// SIMATIC S7-200 SMART project (STEP 7-Micro/WIN SMART), CPU SR30

SYMBOL_TABLE 风机和阀
温度量程下限           VD232
温度量程上限           VD228
压力量程下限           VD324
压力量程上限           VD328
风机停止             V2.0
风机启动             V2.1
风机远程             V2.2
风机故障             V2.3
风机输出             V2.4
风机               V2.5
风机运行反馈           V2.6
风机超时             V2.7
阀1停止             V3.0
阀1启动             V3.1
阀1远程             V3.2
阀1故障             V3.3
阀1输出             V3.4
阀1               V3.5
阀1运行反馈           V3.6
阀1超时             V3.7
阀2停止             V4.0
阀2启动             V4.1
阀2远程             V4.2
阀2故障             V4.3
阀2输出             V4.4
阀2               V4.5
阀2运行反馈           V4.6
阀2超时             V4.7
阀3停止             V5.0
阀3启动             V5.1
阀3远程             V5.2
阀3故障             V5.3
阀3输出             V5.4
阀3               V5.5
阀3运行反馈           V5.6
阀3超时             V5.7
阀4停止             V6.0
阀4启动             V6.1
阀4远程             V6.2
阀4故障             V6.3
阀4输出             V6.4
阀4               V6.5
阀4运行反馈           V6.6
阀4超时             V6.7
END_SYMBOL_TABLE

SYMBOL_TABLE 系统符号
Always_On        SM0.0    // 始终接通
END_SYMBOL_TABLE

SYMBOL_TABLE 点火烧嘴
急停               V10.7
点亮屏幕             V11.1
故障码              VW200
高温报警             V11.2
低温报警             V11.3
流量高报警            V11.4
流量低报警            V11.5
点火命令1            V7.0
点火成功信号1          V7.1
故障复位             V7.2
点火变压器1           V7.3
点火电磁阀1           V7.4
报警1              V7.5
空气压力1            V9.0
燃气压力1            V9.1
燃气泄漏             V9.2
允许点火1            V9.3
本地               V9.4
远程               V9.5
灯光报警1            V10.1
消音自锁             V10.2
声响报警1            V10.3
消音命令             V10.4
点火命令2            V7.6
点火成功信号2          V7.7
点火变压器2           V8.1
点火电磁阀2           V8.2
报警2              V8.3
空气压力2            V9.6
燃气压力2            V9.7
允许点火2            V10.0
灯光报警2            V10.5
声响报警2            V10.6
END_SYMBOL_TABLE

ORGANIZATION_BLOCK MAIN:OB1
TITLE=程序注释
BEGIN
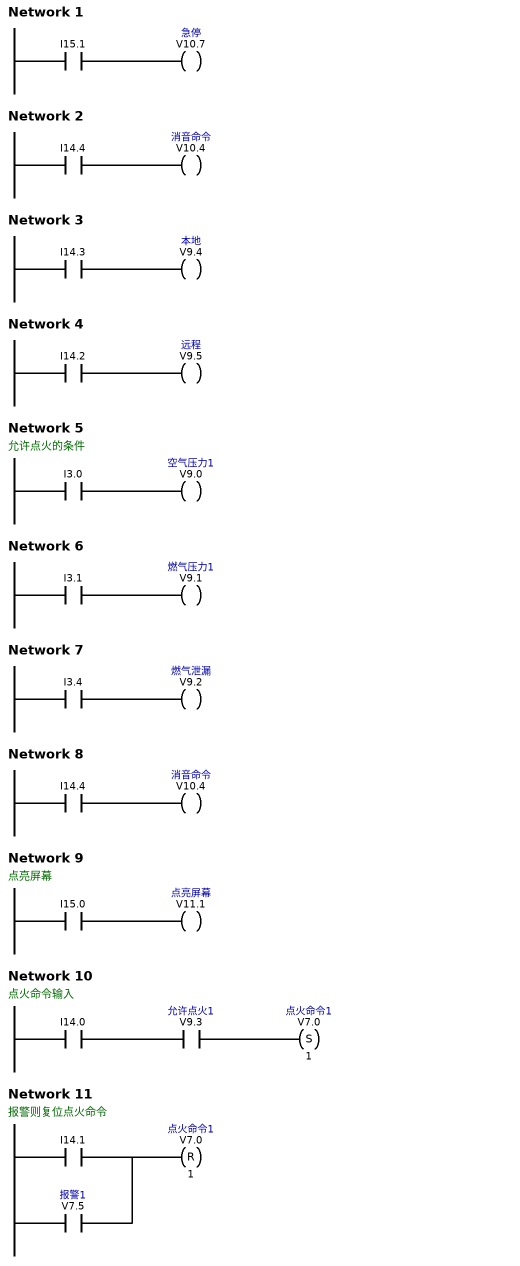
Network 1
LD     I15.1
=      急停:V10.7
Network 2
LD     I14.4
=      消音命令:V10.4
Network 3
LD     I14.3
=      本地:V9.4
Network 4
LD     I14.2
=      远程:V9.5
Network 5
// 允许点火的条件
LD     I3.0
=      空气压力1:V9.0
Network 6
LD     I3.1
=      燃气压力1:V9.1
Network 7
LD     I3.4
=      燃气泄漏:V9.2
Network 8
LD     I14.4
=      消音命令:V10.4
Network 9
// 点亮屏幕
LD     I15.0
=      点亮屏幕:V11.1
Network 10
// 点火命令输入
LD     I14.0
A      允许点火1:V9.3
S      点火命令1:V7.0, 1
Network 11
// 报警则复位点火命令
LD     I14.1
O      报警1:V7.5
R      点火命令1:V7.0, 1
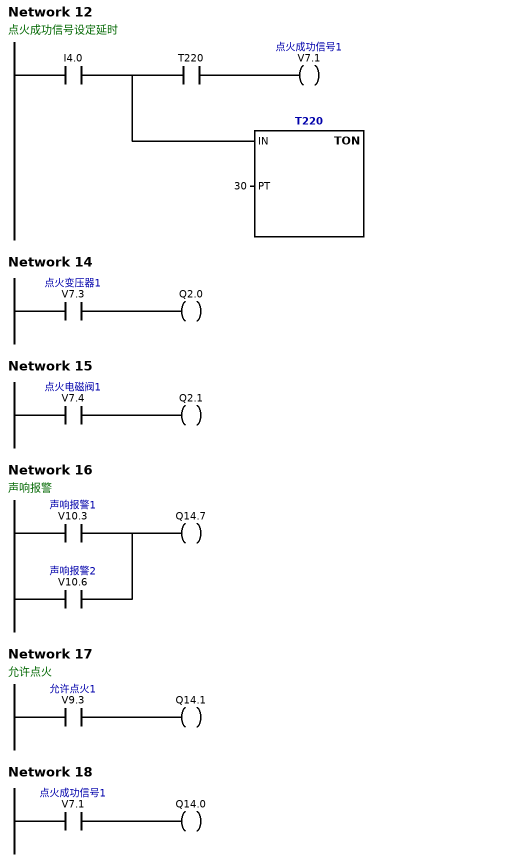
Network 12
// 点火成功信号设定延时
LD     I4.0
LPS
A      T220
=      点火成功信号1:V7.1
LPP
TON    T220, 30
Network 14
LD     点火变压器1:V7.3
=      Q2.0
Network 15
LD     点火电磁阀1:V7.4
=      Q2.1
Network 16
// 声响报警
LD     声响报警1:V10.3
O      声响报警2:V10.6
=      Q14.7
Network 17
// 允许点火
LD     允许点火1:V9.3
=      Q14.1
Network 18
LD     点火成功信号1:V7.1
=      Q14.0
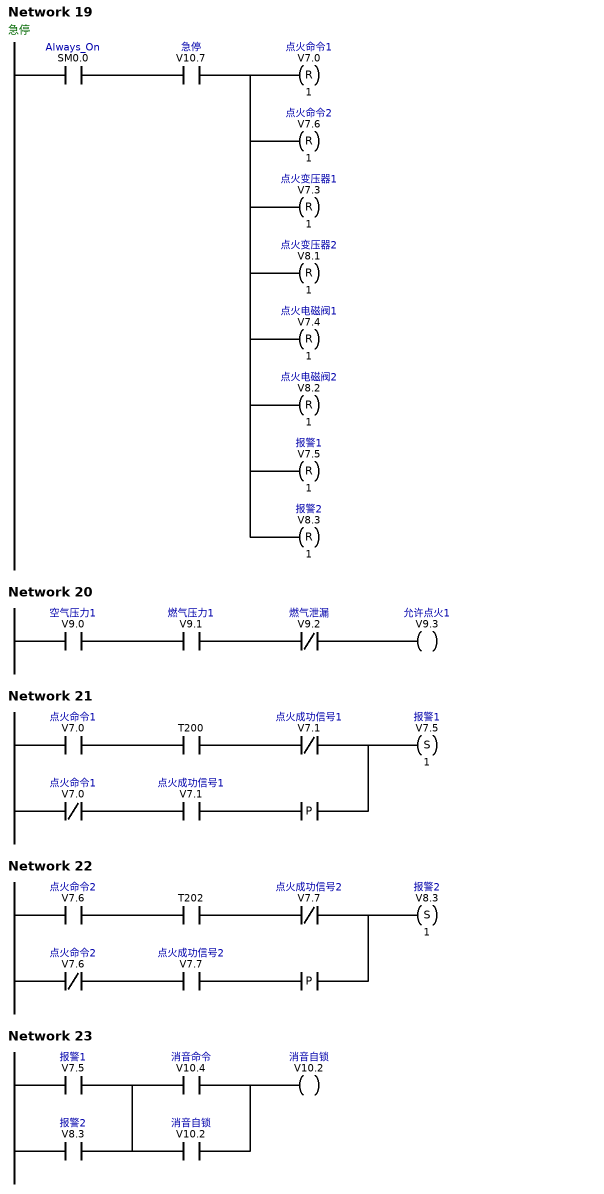
Network 19
// 急停
LD     Always_On:SM0.0
A      急停:V10.7
R      点火命令1:V7.0, 1
R      点火命令2:V7.6, 1
R      点火变压器1:V7.3, 1
R      点火变压器2:V8.1, 1
R      点火电磁阀1:V7.4, 1
R      点火电磁阀2:V8.2, 1
R      报警1:V7.5, 1
R      报警2:V8.3, 1
Network 20
LD     空气压力1:V9.0
A      燃气压力1:V9.1
AN     燃气泄漏:V9.2
=      允许点火1:V9.3
Network 21
LD     点火命令1:V7.0
A      T200
AN     点火成功信号1:V7.1
LDN    点火命令1:V7.0
A      点火成功信号1:V7.1
EU
OLD
S      报警1:V7.5, 1
Network 22
LD     点火命令2:V7.6
A      T202
AN     点火成功信号2:V7.7
LDN    点火命令2:V7.6
A      点火成功信号2:V7.7
EU
OLD
S      报警2:V8.3, 1
Network 23
LD     报警1:V7.5
O      报警2:V8.3
LD     消音命令:V10.4
O      消音自锁:V10.2
ALD
=      消音自锁:V10.2
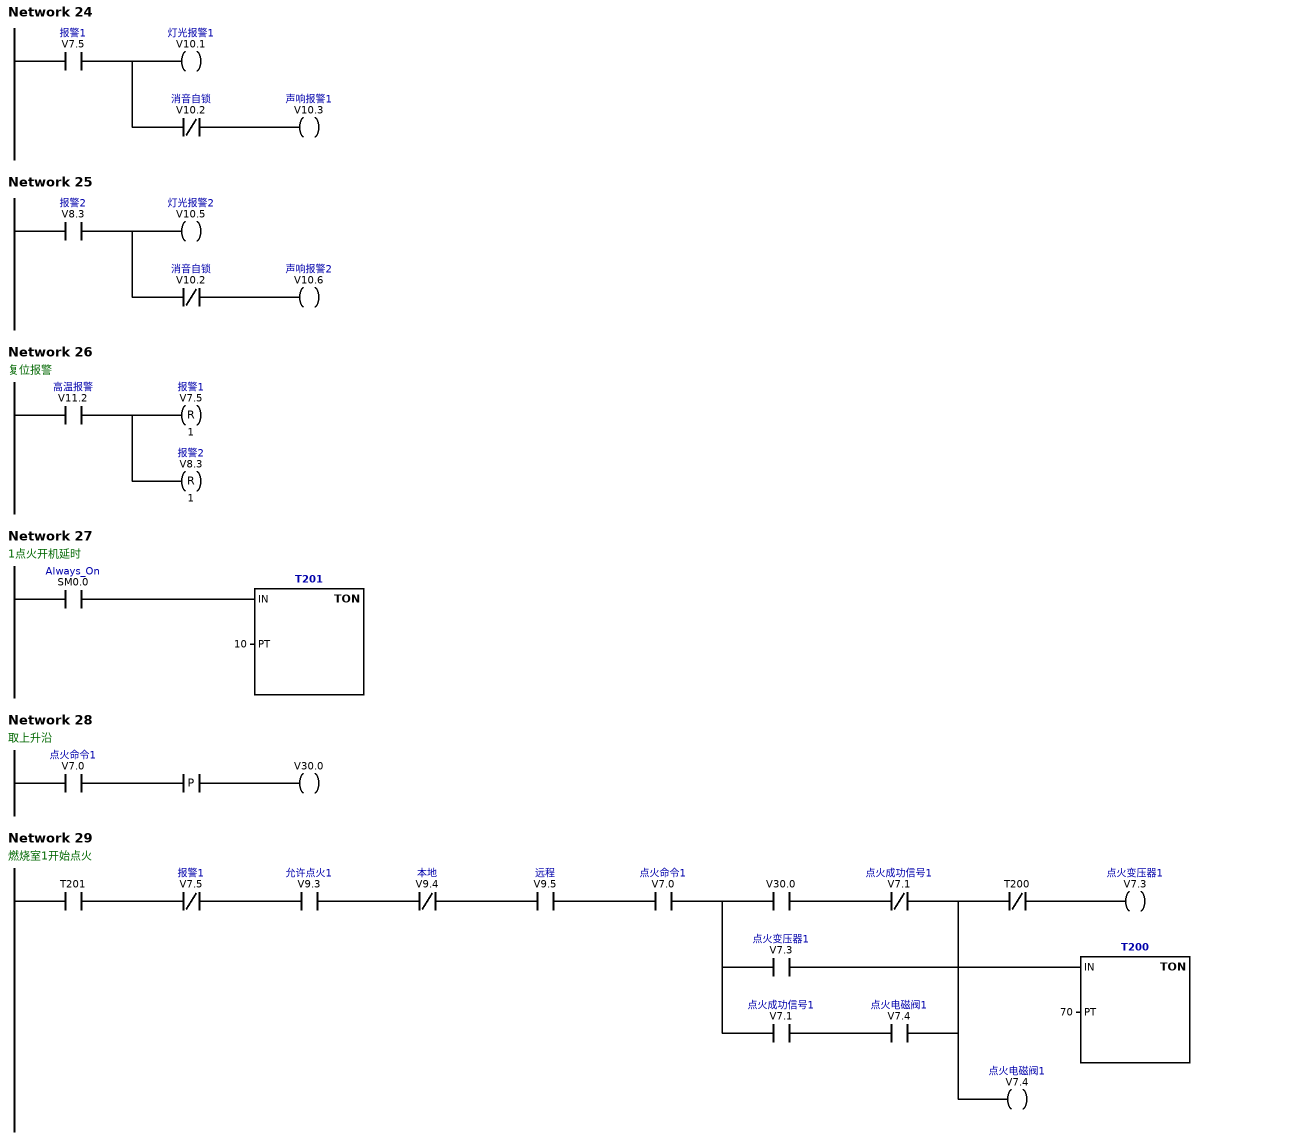
Network 24
LD     报警1:V7.5
=      灯光报警1:V10.1
AN     消音自锁:V10.2
=      声响报警1:V10.3
Network 25
LD     报警2:V8.3
=      灯光报警2:V10.5
AN     消音自锁:V10.2
=      声响报警2:V10.6
Network 26
// 复位报警
LD     高温报警:V11.2
R      报警1:V7.5, 1
R      报警2:V8.3, 1
Network 27
// 1点火开机延时
LD     Always_On:SM0.0
TON    T201, 10
Network 28
// 取上升沿
LD     点火命令1:V7.0
EU
=      V30.0
Network 29
// 燃烧室1开始点火
LD     T201
AN     报警1:V7.5
A      允许点火1:V9.3
AN     本地:V9.4
A      远程:V9.5
A      点火命令1:V7.0
LD     V30.0
AN     点火成功信号1:V7.1
O      点火变压器1:V7.3
LD     点火成功信号1:V7.1
A      点火电磁阀1:V7.4
OLD
ALD
LPS
AN     T200
=      点火变压器1:V7.3
LRD
TON    T200, 70
LPP
=      点火电磁阀1:V7.4
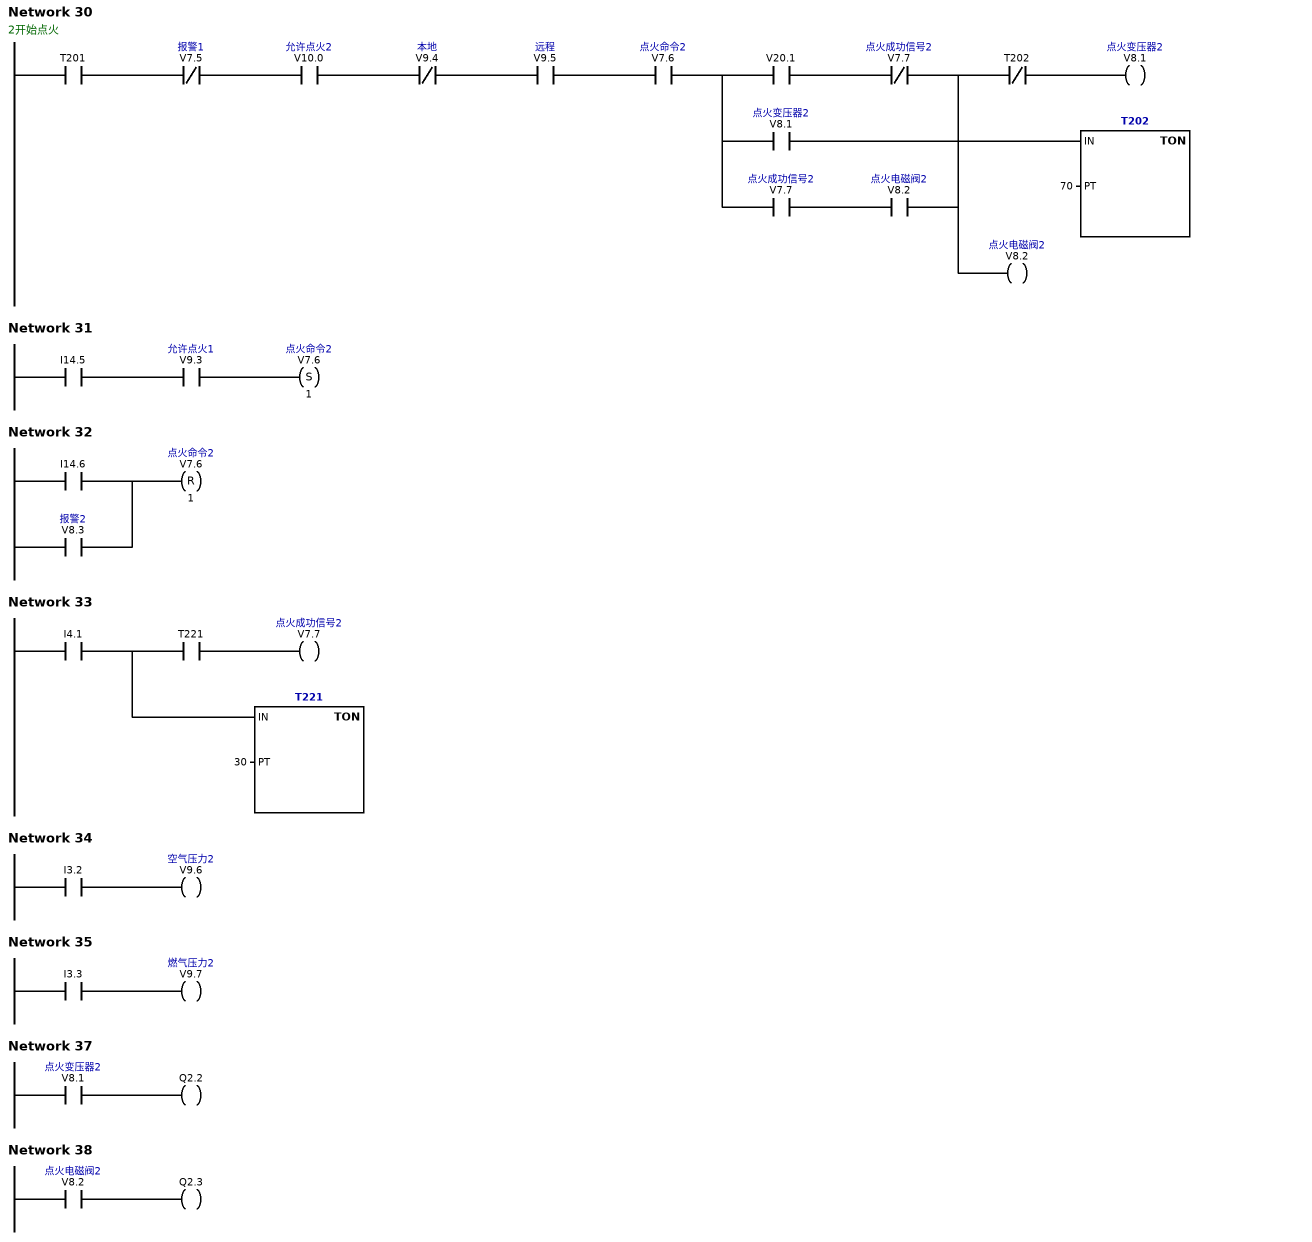
Network 30
// 2开始点火
LD     T201
AN     报警1:V7.5
A      允许点火2:V10.0
AN     本地:V9.4
A      远程:V9.5
A      点火命令2:V7.6
LD     V20.1
AN     点火成功信号2:V7.7
O      点火变压器2:V8.1
LD     点火成功信号2:V7.7
A      点火电磁阀2:V8.2
OLD
ALD
LPS
AN     T202
=      点火变压器2:V8.1
LRD
TON    T202, 70
LPP
=      点火电磁阀2:V8.2
Network 31
LD     I14.5
A      允许点火1:V9.3
S      点火命令2:V7.6, 1
Network 32
LD     I14.6
O      报警2:V8.3
R      点火命令2:V7.6, 1
Network 33
LD     I4.1
LPS
A      T221
=      点火成功信号2:V7.7
LPP
TON    T221, 30
Network 34
LD     I3.2
=      空气压力2:V9.6
Network 35
LD     I3.3
=      燃气压力2:V9.7
Network 37
LD     点火变压器2:V8.1
=      Q2.2
Network 38
LD     点火电磁阀2:V8.2
=      Q2.3
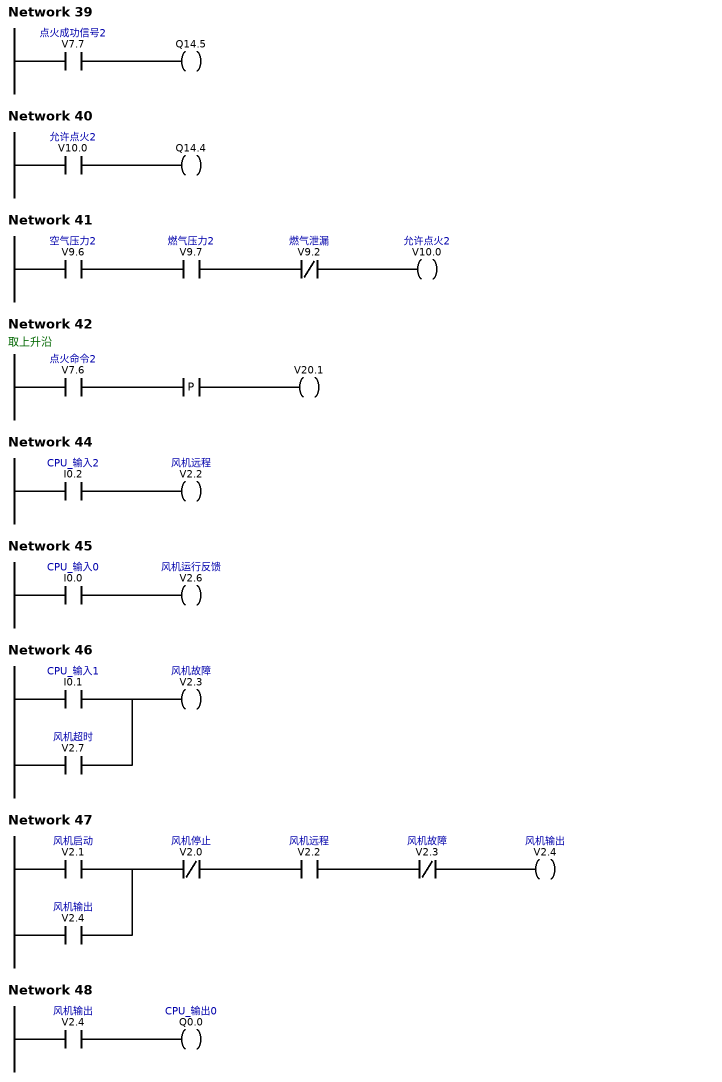
Network 39
LD     点火成功信号2:V7.7
=      Q14.5
Network 40
LD     允许点火2:V10.0
=      Q14.4
Network 41
LD     空气压力2:V9.6
A      燃气压力2:V9.7
AN     燃气泄漏:V9.2
=      允许点火2:V10.0
Network 42
// 取上升沿
LD     点火命令2:V7.6
EU
=      V20.1
Network 44
LD     CPU_输入2:I0.2
=      风机远程:V2.2
Network 45
LD     CPU_输入0:I0.0
=      风机运行反馈:V2.6
Network 46
LD     CPU_输入1:I0.1
O      风机超时:V2.7
=      风机故障:V2.3
Network 47
LD     风机启动:V2.1
O      风机输出:V2.4
AN     风机停止:V2.0
A      风机远程:V2.2
AN     风机故障:V2.3
=      风机输出:V2.4
Network 48
LD     风机输出:V2.4
=      CPU_输出0:Q0.0
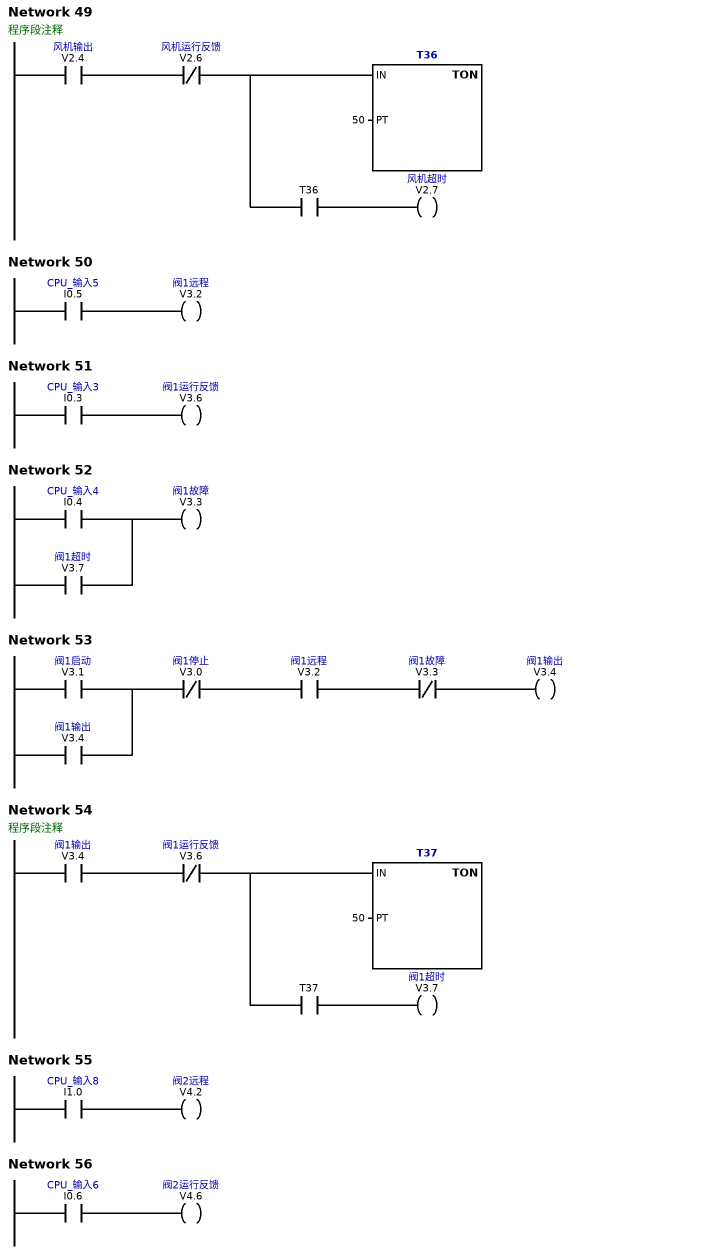
Network 49
// 程序段注释
LD     风机输出:V2.4
AN     风机运行反馈:V2.6
TON    T36, 50
A      T36
=      风机超时:V2.7
Network 50
LD     CPU_输入5:I0.5
=      阀1远程:V3.2
Network 51
LD     CPU_输入3:I0.3
=      阀1运行反馈:V3.6
Network 52
LD     CPU_输入4:I0.4
O      阀1超时:V3.7
=      阀1故障:V3.3
Network 53
LD     阀1启动:V3.1
O      阀1输出:V3.4
AN     阀1停止:V3.0
A      阀1远程:V3.2
AN     阀1故障:V3.3
=      阀1输出:V3.4
Network 54
// 程序段注释
LD     阀1输出:V3.4
AN     阀1运行反馈:V3.6
TON    T37, 50
A      T37
=      阀1超时:V3.7
Network 55
LD     CPU_输入8:I1.0
=      阀2远程:V4.2
Network 56
LD     CPU_输入6:I0.6
=      阀2运行反馈:V4.6
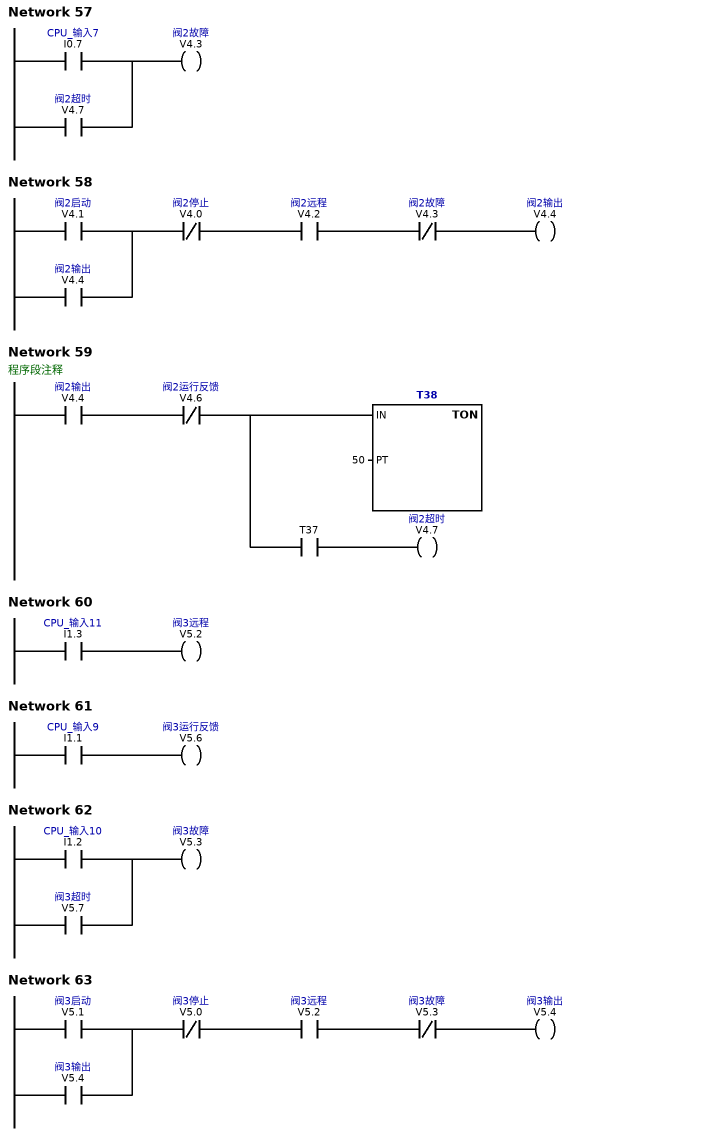
Network 57
LD     CPU_输入7:I0.7
O      阀2超时:V4.7
=      阀2故障:V4.3
Network 58
LD     阀2启动:V4.1
O      阀2输出:V4.4
AN     阀2停止:V4.0
A      阀2远程:V4.2
AN     阀2故障:V4.3
=      阀2输出:V4.4
Network 59
// 程序段注释
LD     阀2输出:V4.4
AN     阀2运行反馈:V4.6
TON    T38, 50
A      T37
=      阀2超时:V4.7
Network 60
LD     CPU_输入11:I1.3
=      阀3远程:V5.2
Network 61
LD     CPU_输入9:I1.1
=      阀3运行反馈:V5.6
Network 62
LD     CPU_输入10:I1.2
O      阀3超时:V5.7
=      阀3故障:V5.3
Network 63
LD     阀3启动:V5.1
O      阀3输出:V5.4
AN     阀3停止:V5.0
A      阀3远程:V5.2
AN     阀3故障:V5.3
=      阀3输出:V5.4
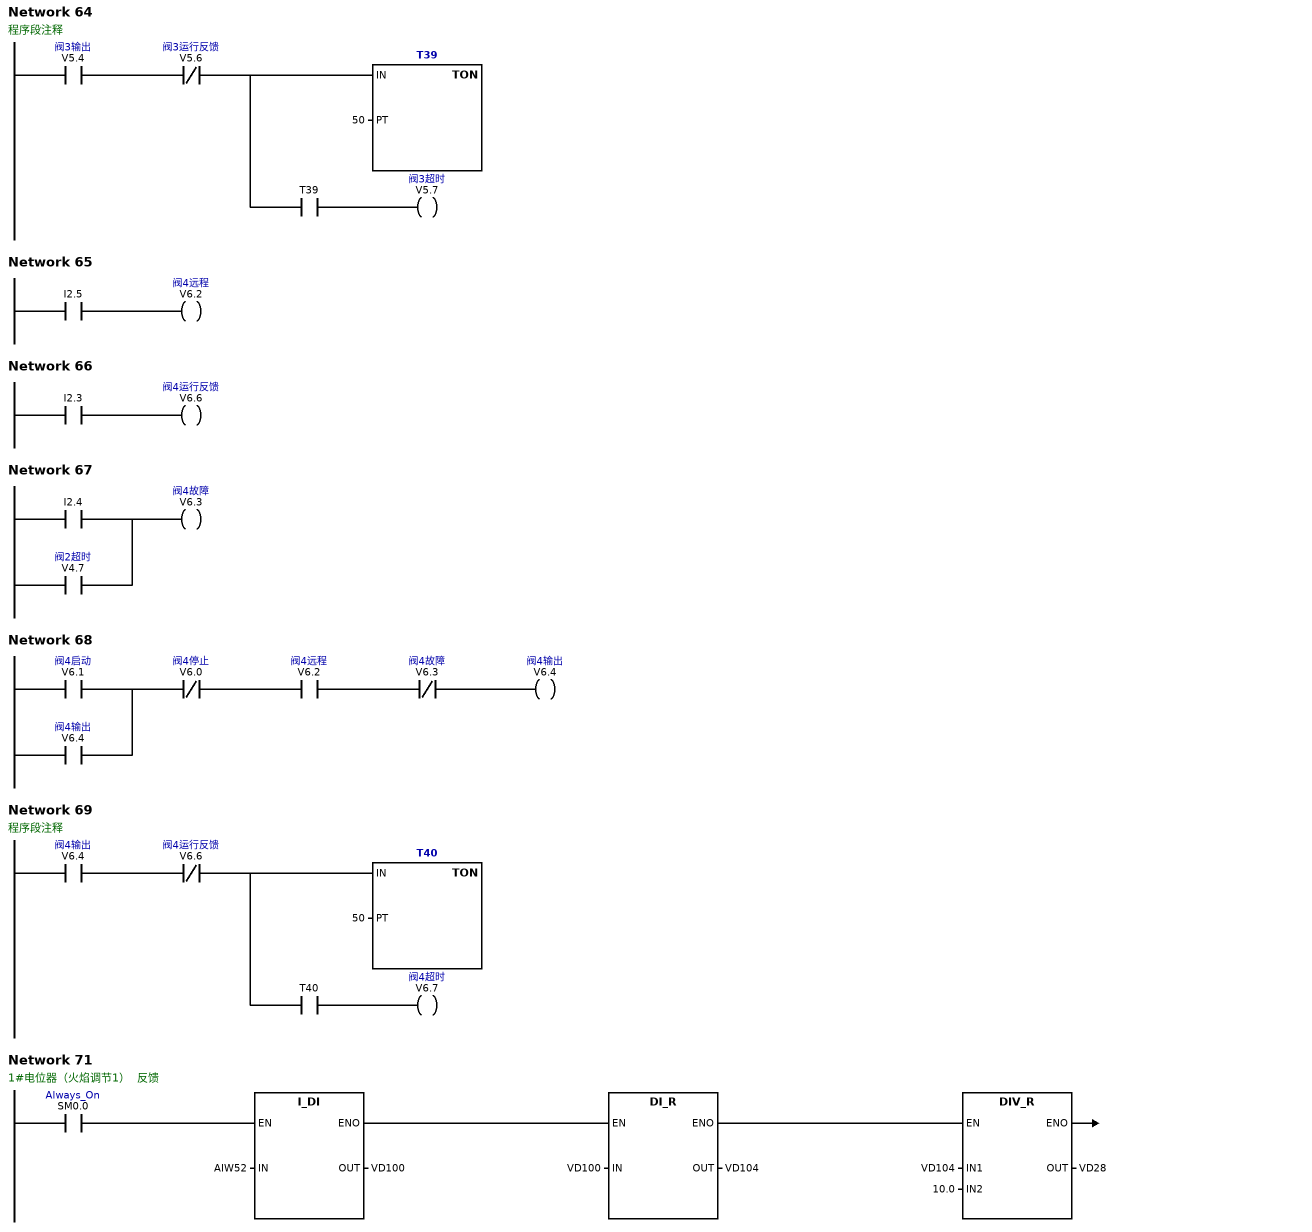
Network 64
// 程序段注释
LD     阀3输出:V5.4
AN     阀3运行反馈:V5.6
TON    T39, 50
A      T39
=      阀3超时:V5.7
Network 65
LD     I2.5
=      阀4远程:V6.2
Network 66
LD     I2.3
=      阀4运行反馈:V6.6
Network 67
LD     I2.4
O      阀2超时:V4.7
=      阀4故障:V6.3
Network 68
LD     阀4启动:V6.1
O      阀4输出:V6.4
AN     阀4停止:V6.0
A      阀4远程:V6.2
AN     阀4故障:V6.3
=      阀4输出:V6.4
Network 69
// 程序段注释
LD     阀4输出:V6.4
AN     阀4运行反馈:V6.6
TON    T40, 50
A      T40
=      阀4超时:V6.7
Network 71
// 1#电位器（火焰调节1）  反馈
LD     Always_On:SM0.0
ITD    AIW52, VD100
AENO
DTR    VD100, VD104
AENO
MOVR   VD104, VD28
/R     10.0, VD28
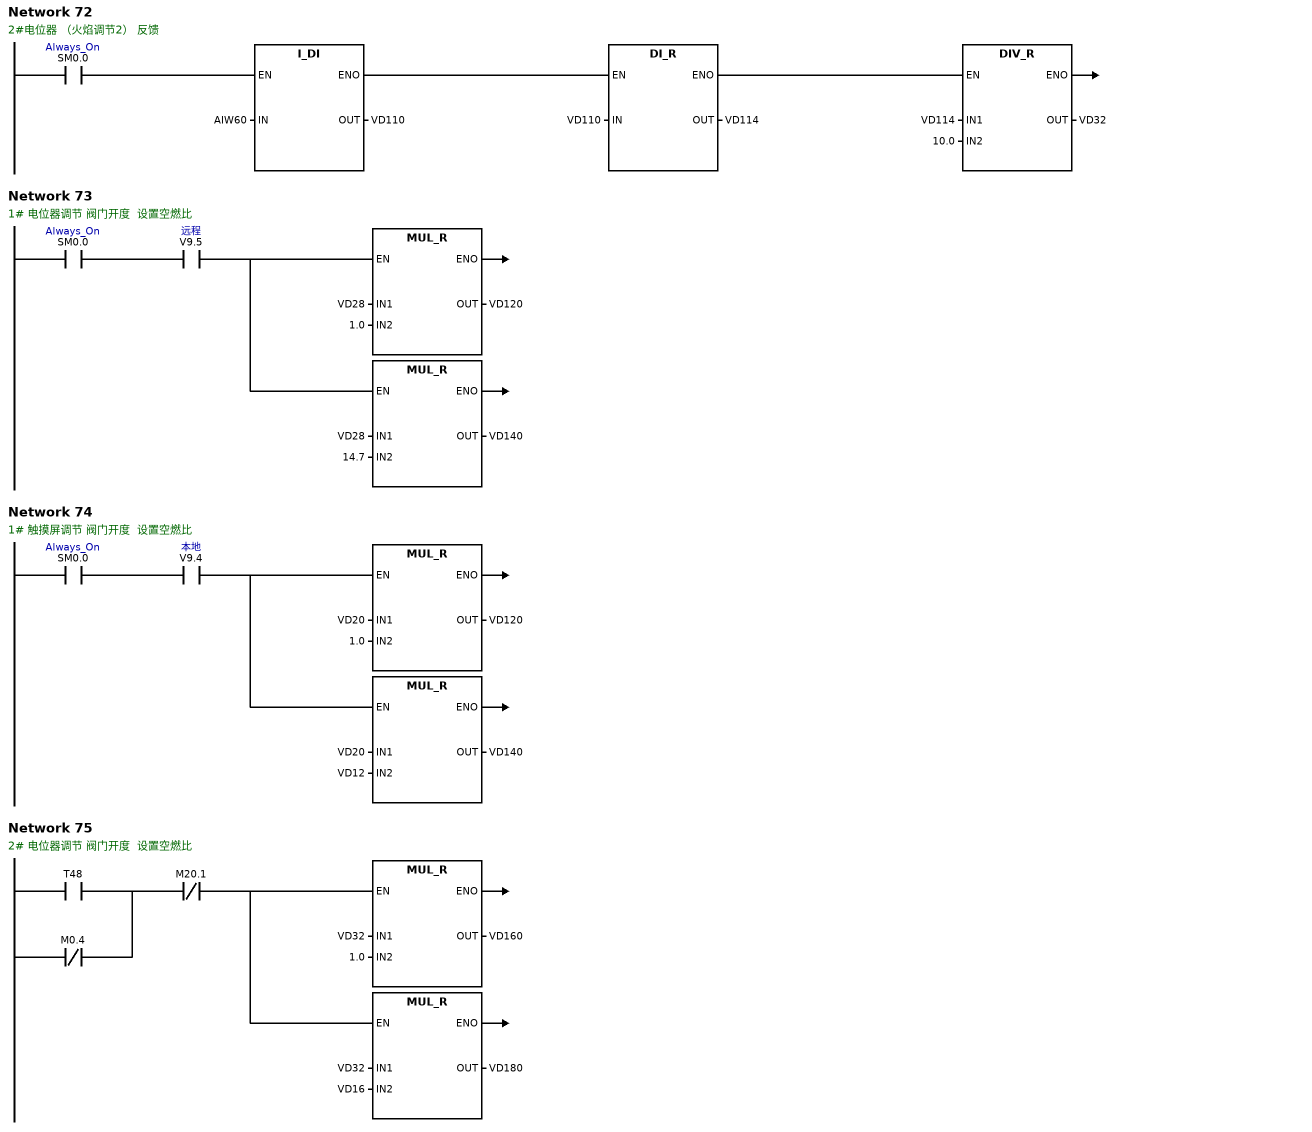
Network 72
// 2#电位器 （火焰调节2） 反馈
LD     Always_On:SM0.0
ITD    AIW60, VD110
AENO
DTR    VD110, VD114
AENO
MOVR   VD114, VD32
/R     10.0, VD32
Network 73
// 1# 电位器调节 阀门开度  设置空燃比
LD     Always_On:SM0.0
A      远程:V9.5
MOVR   VD28, VD120
*R     1.0, VD120
MOVR   VD28, VD140
*R     14.7, VD140
Network 74
// 1# 触摸屏调节 阀门开度  设置空燃比
LD     Always_On:SM0.0
A      本地:V9.4
MOVR   VD20, VD120
*R     1.0, VD120
MOVR   VD20, VD140
*R     VD12, VD140
Network 75
// 2# 电位器调节 阀门开度  设置空燃比
LD     T48
ON     M0.4
AN     M20.1
MOVR   VD32, VD160
*R     1.0, VD160
MOVR   VD32, VD180
*R     VD16, VD180
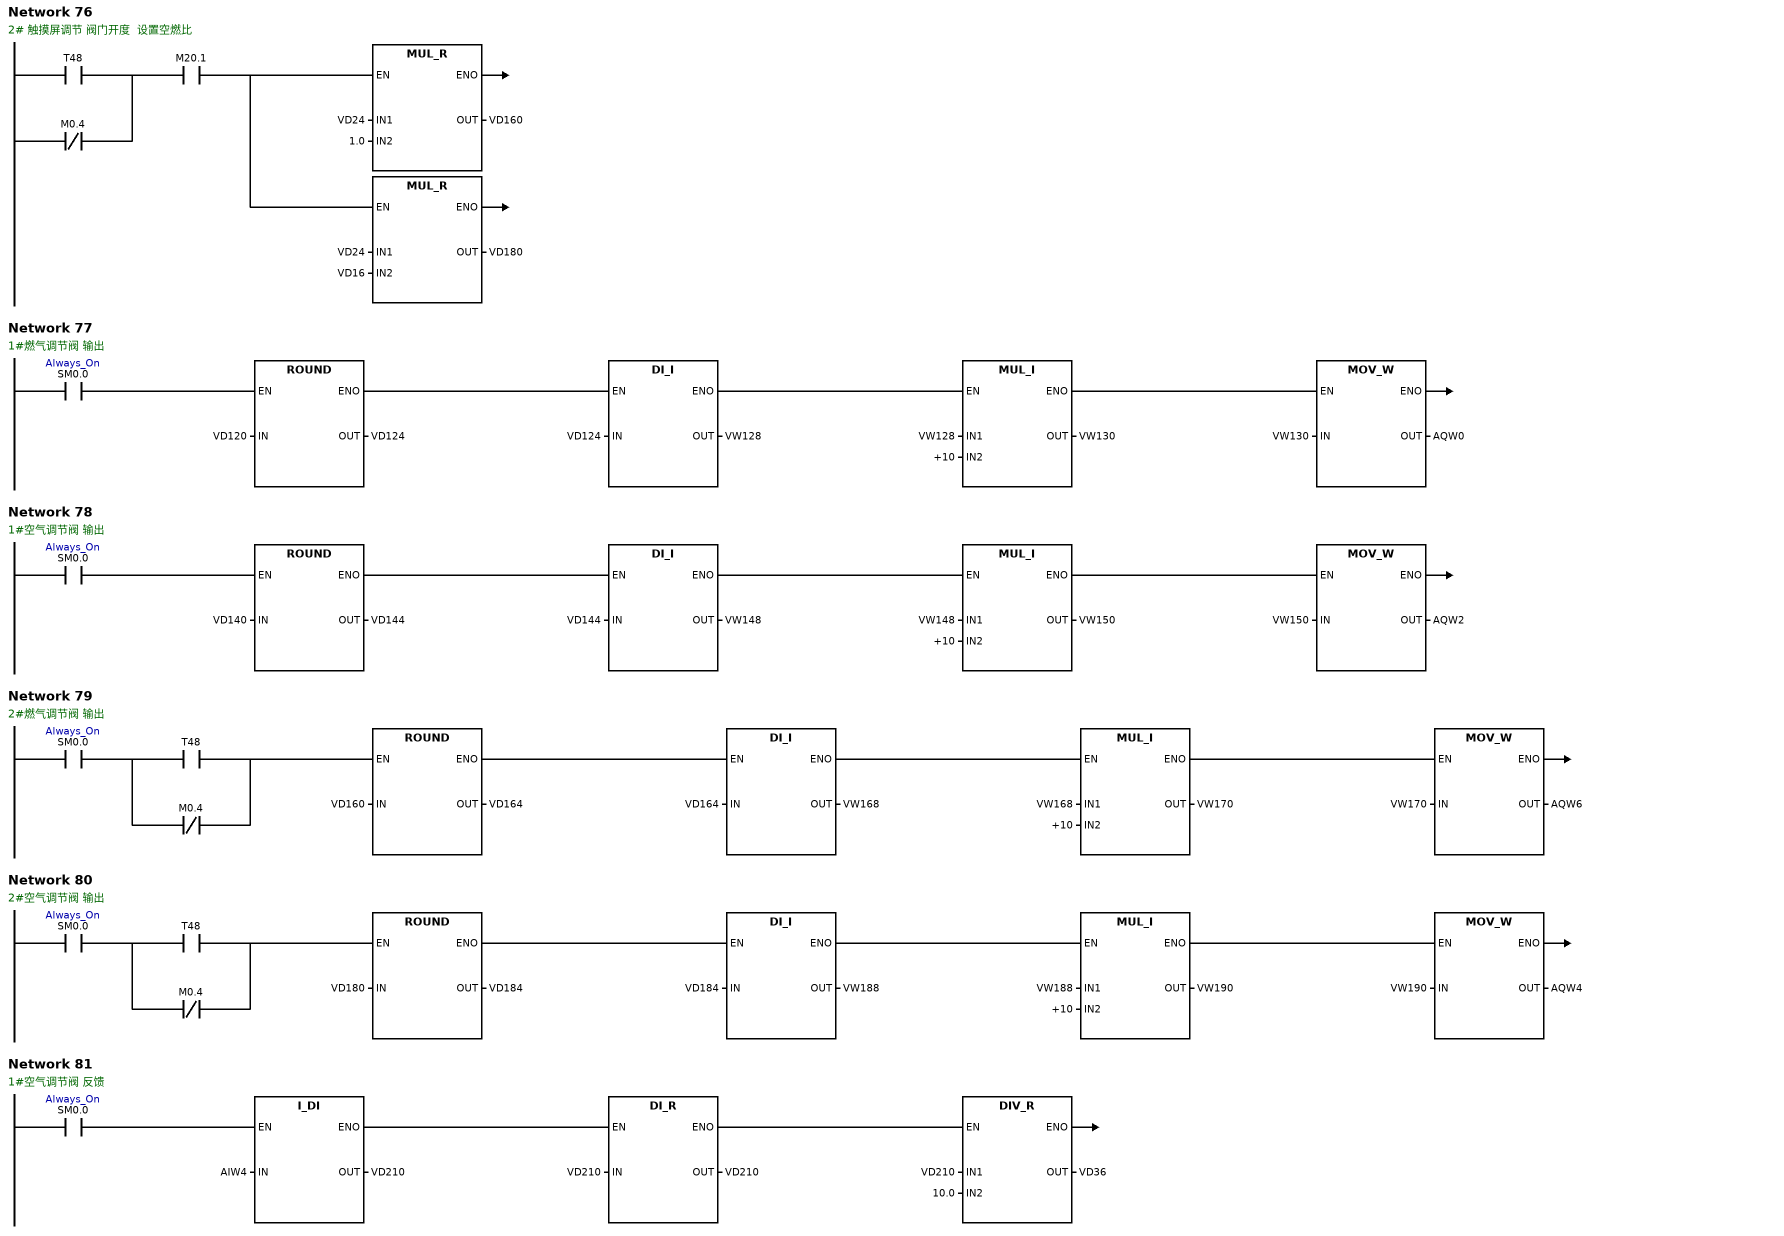
Network 76
// 2# 触摸屏调节 阀门开度  设置空燃比
LD     T48
ON     M0.4
A      M20.1
MOVR   VD24, VD160
*R     1.0, VD160
MOVR   VD24, VD180
*R     VD16, VD180
Network 77
// 1#燃气调节阀 输出
LD     Always_On:SM0.0
ROUND  VD120, VD124
AENO
DTI    VD124, VW128
AENO
MOVW   VW128, VW130
AENO
*I     +10, VW130
AENO
MOVW   VW130, AQW0
Network 78
// 1#空气调节阀 输出
LD     Always_On:SM0.0
ROUND  VD140, VD144
AENO
DTI    VD144, VW148
AENO
MOVW   VW148, VW150
AENO
*I     +10, VW150
AENO
MOVW   VW150, AQW2
Network 79
// 2#燃气调节阀 输出
LD     Always_On:SM0.0
LD     T48
ON     M0.4
ALD
ROUND  VD160, VD164
AENO
DTI    VD164, VW168
AENO
MOVW   VW168, VW170
AENO
*I     +10, VW170
AENO
MOVW   VW170, AQW6
Network 80
// 2#空气调节阀 输出
LD     Always_On:SM0.0
LD     T48
ON     M0.4
ALD
ROUND  VD180, VD184
AENO
DTI    VD184, VW188
AENO
MOVW   VW188, VW190
AENO
*I     +10, VW190
AENO
MOVW   VW190, AQW4
Network 81
// 1#空气调节阀 反馈
LD     Always_On:SM0.0
ITD    AIW4, VD210
AENO
DTR    VD210, VD210
AENO
MOVR   VD210, VD36
/R     10.0, VD36
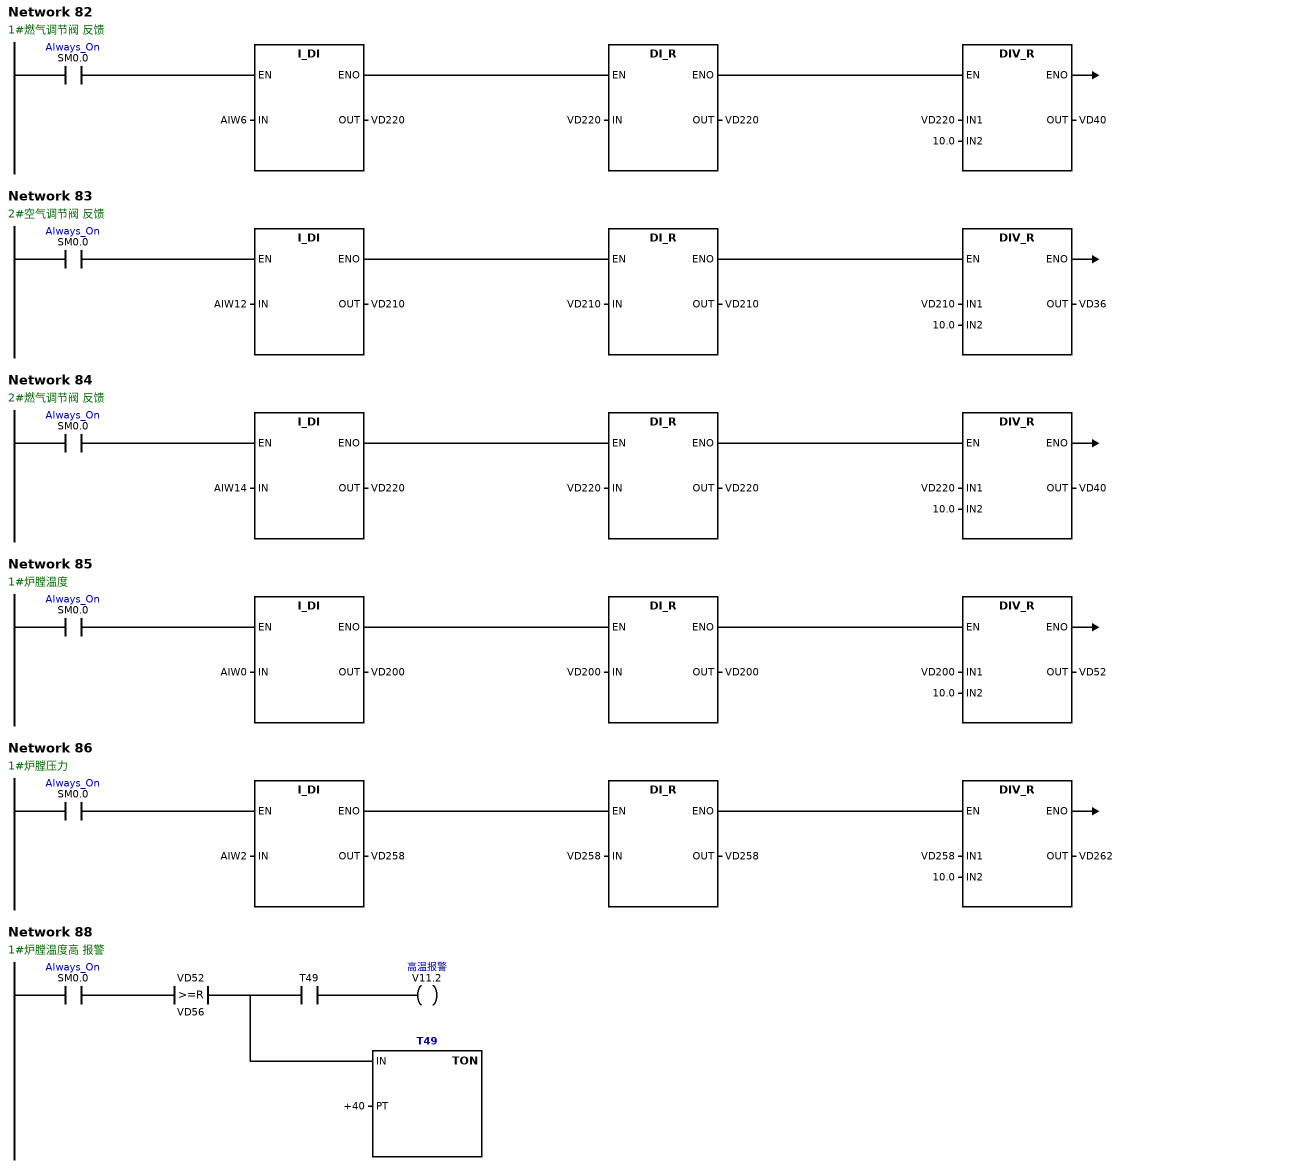
Network 82
// 1#燃气调节阀 反馈
LD     Always_On:SM0.0
ITD    AIW6, VD220
AENO
DTR    VD220, VD220
AENO
MOVR   VD220, VD40
/R     10.0, VD40
Network 83
// 2#空气调节阀 反馈
LD     Always_On:SM0.0
ITD    AIW12, VD210
AENO
DTR    VD210, VD210
AENO
MOVR   VD210, VD36
/R     10.0, VD36
Network 84
// 2#燃气调节阀 反馈
LD     Always_On:SM0.0
ITD    AIW14, VD220
AENO
DTR    VD220, VD220
AENO
MOVR   VD220, VD40
/R     10.0, VD40
Network 85
// 1#炉膛温度
LD     Always_On:SM0.0
ITD    AIW0, VD200
AENO
DTR    VD200, VD200
AENO
MOVR   VD200, VD52
/R     10.0, VD52
Network 86
// 1#炉膛压力
// (network saved uncompiled; LAD cells follow)
// row 0: c0 -| |- Always_On:SM0.0  c1 --  c2 [I_DI EN:=power@row0, IN:=AIW2, ENO=>power, OUT=>VD258]  c3 --  c4 --  c5 [DI_R EN:=power@row0, IN:=VD258, ENO=>power, OUT=>VD258]  c6 --  c7 --  c8 [DIV_R EN:=power@row0, IN1:=VD258, IN2:=10.0, ENO=>power, OUT=>VD262]  c9 ->
// row 1: c2 [box]  c5 [box]  c8 [box]
Network 88
// 1#炉膛温度高 报警
LD     Always_On:SM0.0
AR>=   VD52, VD56
LPS
A      T49
=      高温报警:V11.2
LPP
TON    T49, +40
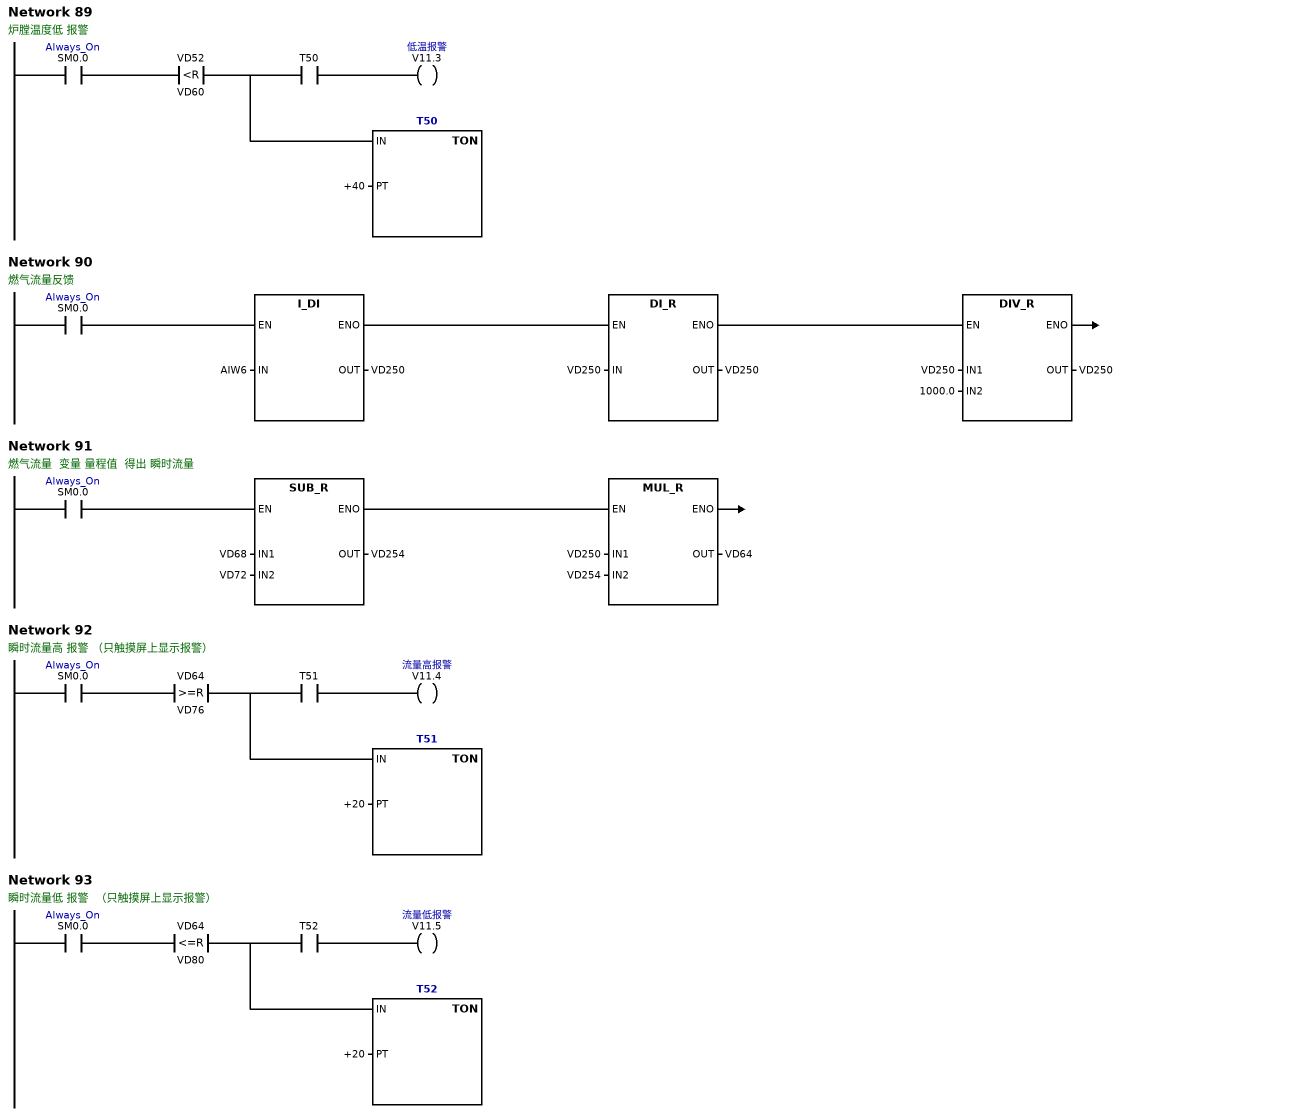
Network 89
// 炉膛温度低 报警
LD     Always_On:SM0.0
AR<    VD52, VD60
LPS
A      T50
=      低温报警:V11.3
LPP
TON    T50, +40
Network 90
// 燃气流量反馈
LD     Always_On:SM0.0
ITD    AIW6, VD250
AENO
DTR    VD250, VD250
AENO
/R     1000.0, VD250
Network 91
// 燃气流量  变量 量程值  得出 瞬时流量
LD     Always_On:SM0.0
MOVR   VD68, VD254
AENO
-R     VD72, VD254
AENO
MOVR   VD250, VD64
*R     VD254, VD64
Network 92
// 瞬时流量高 报警 （只触摸屏上显示报警）
LD     Always_On:SM0.0
AR>=   VD64, VD76
LPS
A      T51
=      流量高报警:V11.4
LPP
TON    T51, +20
Network 93
// 瞬时流量低 报警  （只触摸屏上显示报警）
LD     Always_On:SM0.0
AR<=   VD64, VD80
LPS
A      T52
=      流量低报警:V11.5
LPP
TON    T52, +20
END_ORGANIZATION_BLOCK

// SBR1: protected block, not included

// SBR2: protected block, not included

// SBR3: protected block, not included

// SBR4: protected block, not included

// SBR5: protected block, not included

// SBR6: protected block, not included

// SBR7: protected block, not included
